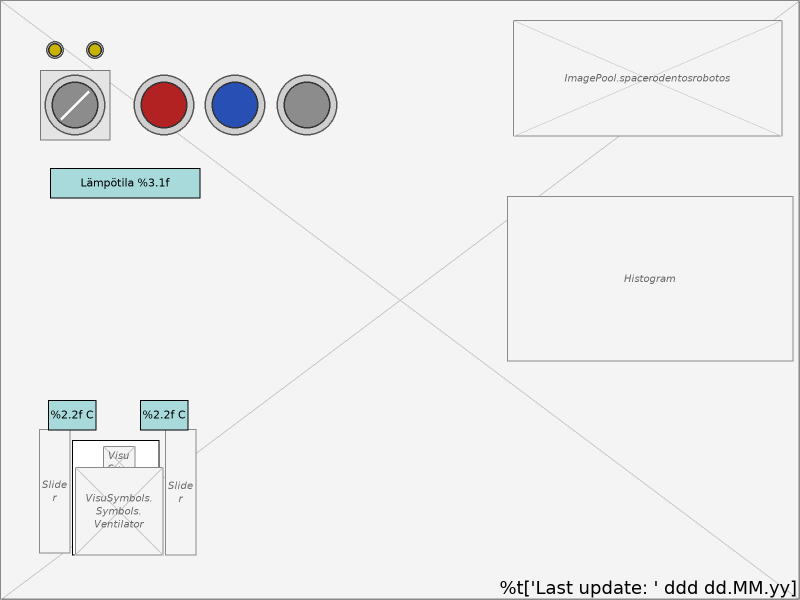
VISUALIZATION Visualization  // 800x600
    Image (0,0 800x600), "%t['Last update: ' ddd dd.MM.yy]", image: ImagePool.PLC UI 10
    Lamp1 (129,70 70x70), variable: IO.out_punainenvalo, style: Lamp-Lamp1-Red
    Lamp1 (200,70 70x70), variable: IO.out_sininenvalo, style: Lamp-Lamp1-Blue
    Lamp1 (272,70 70x70), variable: IO.out_valkoinenvalo, style: Lamp-Lamp1-Gray
    RoundedRectangle (50,168 150x30), "Lämpötila %3.1f", text variable: Lampotilailu.lampotila_decimaalit
    Histogram (507,196 286x165), scale format: %.1f, scale 150..350
        p1518820177: ui.aLampo
        p102497268: ui.aLampo
        p788070771: ARRAY [1..10] OF INT
    Image (513,20 269x116), image: ImagePool.spacerodentosrobotos
    RotarySwitch (40,70 70x70), behaviour: TOGGLE, style: Switch-RotarySwitch-Gray
    Lamp1 (45,40 20x20), variable: IO.in_vipu_vasen, style: Lamp-Lamp1-Yellow
    Lamp1 (85,40 20x20), variable: IO.in_vipu_oikea, style: Lamp-Lamp1-Yellow
    Group (72,440 91x115)
        RoundedRectangle (0,0 87x115), colour toggle: IO.out_tuuletin, colour variable: 16#FF457B9D
            p2167032090: 16#FF8FE03F
        Image (31,6 32x32), colour toggle: IO.out_tuuletin, image: VisuSymbols.Symbols.ArrowHalfRightRight
            p2175578022: 16#FF1DC85A
            p573394764: 16#FF791426
        Image (3,27 88x88), image: VisuSymbols.Symbols.Ventilator
    Slider (165,429 31x126), variable: ui.TEMP_HI_LIMIT, scale 200..270
    Slider (39,429 31x124), variable: ui.TEMP_LO_LIMIT, scale 150..270
    RoundedRectangle (140,400 48x30), "%2.2f C", text variable: Lampotilailu.TEMP_HI_DECIMAL
    RoundedRectangle (48,400 48x30), "%2.2f C", text variable: Lampotilailu.TEMP_LO_DECIMAL
END_VISUALIZATION

(* stored: Version 1.1.0.1, ProductVersion 3.1.4024.6
   Visu Visualization: Id {57f422e5-be05-4061-9c76-5d6e41674097} *)
